Staubli VAL3: HIT_YD.pjx

--- HIT_YD.pjx ---
Parameters version=s7.6.2 stackSize=5000 millimeterUnit=true
Program file=OMAC_Abort.pgx
Program file=OMAC_Hold.pgx
Program file=OMAC_Main.pgx
Program file=OMAC_Reset.pgx
Program file=OMAC_Start.pgx
Program file=OMAC_Stop.pgx
Program file=OMAC_Unhold.pgx
Program file=blow.pgx
Program file=bypassPick.pgx
Program file=cellManager.pgx
Program file=getToolStatus.pgx
Program file=goHome.pgx
Program file=init.pgx
Program file=initTracking.pgx
Program file=isInSafetyArea.pgx
Program file=ModbusGet.pgx
Program file=modbusSet.pgx
Program file=overflowPick.pgx
Program file=Place.pgx
Program file=productionCycle.pgx
Program file=robot2PC.pgx
Program file=robot2PLC.pgx
Program file=send2NextRob.pgx
Program file=setAlarm.pgx
Program file=setConvSpeed.pgx
Program file=start.pgx
Program file=stop.pgx
Program file=trackErr_init.pgx
Program file=trackingPick.pgx
Program file=transferQueue.pgx
Data file=HIT_YD.dtx
Library alias=mot path=Disk://Tracking/Motion/Motion.pjx autoload=true password=
Type name=object path=Disk://Tracking/Templates/object/object.pjx

--- HIT_YD.dtx ---
aio aConvSpeed = {link=ModbusSrv-0\Modbus-Word\ao[3]}
aio aPlcCmd = {link=ModbusSrv-0\Modbus-Word\ai[0]}
aio aRbAlarm = {link=ModbusSrv-0\Modbus-Word\ao[0]}
aio aRbStatus = {link=ModbusSrv-0\Modbus-Word\ao[1]}
bool _bConvExist = true
bool _bEndCycle
bool _bIsPicking = true
bool _bIsPlacing
bool _bMutexCnvQueue = true
bool _bOverflowed = true
bool _bPartInTool
bool _bSentToHome = true
bool _bVisionOK = true
bool bLockPage
bool bPickDetection
bool bSetConvSpeed
bool bSyn
bool bTransferData = true
dio dAlarm[8]
  [0] = {link=ModbusSrv-0\Modbus-Bit\do[8]}
  [1] = {link=ModbusSrv-0\Modbus-Bit\do[9]}
  [2] = {link=ModbusSrv-0\Modbus-Bit\do[10]}
  [3] = {link=ModbusSrv-0\Modbus-Bit\do[11]}
  [4] = {link=ModbusSrv-0\Modbus-Bit\do[12]}
  [5] = {link=ModbusSrv-0\Modbus-Bit\do[13]}
  [6] = {link=ModbusSrv-0\Modbus-Bit\do[14]}
  [7] = {link=ModbusSrv-0\Modbus-Bit\do[15]}
dio dBlow = {link=BasicIO-1\%Q5}
dio dConvControl[2]
  [0] = {link=BasicIO-1\%I4}
  [1] = {link=BasicIO-1\%Q6}
dio dPartInTool = {link=fIn0}
dio dPermitPlace[4]
  [0] = {link=BasicIO-1\%I3}
  [1] = {link=BasicIO-1\%I2}
  [2] = {link=BasicIO-1\%I1}
  [3] = {link=BasicIO-1\%I0}
dio dPlaceDone[4]
  [0] = {link=BasicIO-1\%Q11}
  [1] = {link=BasicIO-1\%Q10}
  [2] = {link=BasicIO-1\%Q9}
  [3] = {link=BasicIO-1\%Q8}
dio dStartControl[4]
  [0] = {link=ModbusSrv-0\Modbus-Bit\di[4]}
  [1] = {link=ModbusSrv-0\Modbus-Bit\di[5]}
  [2] = {link=ModbusSrv-0\Modbus-Bit\di[6]}
  [3] = {link=ModbusSrv-0\Modbus-Bit\di[7]}
dio dStartState[4]
  [0] = {link=ModbusSrv-0\Modbus-Bit\do[4]}
  [1] = {link=ModbusSrv-0\Modbus-Bit\do[5]}
  [2] = {link=ModbusSrv-0\Modbus-Bit\do[6]}
  [3] = {link=ModbusSrv-0\Modbus-Bit\do[7]}
dio dVacuum = {link=BasicIO-1\%Q4}
frame fConveyor = {x=365.904087, y=326.91934, z=-82.602337, rx=-0.010861, ry=-0.059106, rz=0.004608, fatherId=world[0]}
frame fDetection = {x=392.598601, y=461.346273, z=-82.976862, rx=0.205045, ry=0.617271, rz=0.011036, fatherId=world[0]}
jointRs jDropPart = {j1=102.785955, j2=-95.43121, j3=69.578977, j4=134.260732}
jointRs jHome = {j1=102.785955, j2=-95.43121, j3=69.578977, j4=134.260732}
jointRs jPark = {j1=102.785955, j2=-95.43121, j3=69.578977, j4=134.260732}
mdesc _mLoad = {accel=98.01, vel=99, decel=98.01, leave=40, reach=40}
mdesc mLoad = {accel=121, vel=110, decel=121, leave=40, reach=40}
mdesc mNomSpeed = {accel=121, vel=110, decel=121, leave=20, reach=20}
mdesc mPickDown = {accel=144, vel=120, decel=144, blend=off, leave=10, reach=10}
mdesc mPickup = {accel=121, vel=110, decel=121, leave=40, reach=40}
mdesc mPlaceDown = {accel=144, vel=120, decel=144, blend=off, leave=15, reach=15}
mdesc mPlaceUp = {accel=169, vel=130, decel=169, blend=cartesian, leave=30, reach=30}
mdesc mSlow = {accel=1, vel=10, decel=1, leave=10, reach=10}
mdesc mUnload = {accel=121, vel=110, decel=121, leave=40, reach=40}
num _nBlowDelay
num _nCntBypassed = 1
num _nCntPartsDone[2]
  [0] = 234927
  [1] = 234852
num _nCntTransfered = 2732
num _nConvSpd = 482.240758
num _nCycleTime[4]
  [0] = 2.619
  [1] = 0.715
  [2] = 2.425
  [3] = 0.561
num _nCycleTimeIndx = 2
num _nID = 1
num _nLastStateCMD
num _nOmacStat = 3
num _nPartID = 1
num _nPlaceCurItem[2]
num _nPullIndexTQ = 32
num _nPushIndexTQ = 32
num _nStateCMD
num _nTimer = 6773.495
num _nTrackErr = 334
num nBlowID = 0.4
num nBypass = 1
num nLoadRatio[4]
  [0] = 0.85
  [1] = 0.9
  [2] = 0.9
  [3] = 1
num nNomConvSpeed = 100
num nPartHeight = 5
num nPickAppro = 65
num nPickOS_X
num nPickOS_Y = 2
num nPlaceAppro = 60
public num nPlaceNum
num nSafeMaxX = 850
num nSafeMaxY = 650
num nSafeMinX
num nSafeMinY
num nStopTime
num nTestData[5]
  [0] = 6
  [1] = -49
  [2] = 55
  [4] = 184151
num nVacuumID = 0.1
num nWaitDist2Up4BP = -300
num nWaitDistToDown = 50
num nWaitDistToUp[1 3]
  [0,0] = -80
  [0,1] = 120
  [0,2] = 400
num nWaitDistX
object _oTransferQueue[1 100]
  [0,0]
    num nID = -1
    num nLatchedValue
    trsf trTrsf
  [0,1]
    num nID = -1
    num nLatchedValue
    trsf trTrsf
  [0,2]
    num nID = -1
    num nLatchedValue
    trsf trTrsf
  [0,3]
    num nID = -1
    num nLatchedValue
    trsf trTrsf
  [0,4]
    num nID = -1
    num nLatchedValue
    trsf trTrsf
  [0,5]
    num nID = -1
    num nLatchedValue
    trsf trTrsf
  [0,6]
    num nID = -1
    num nLatchedValue
    trsf trTrsf
  [0,7]
    num nID = -1
    num nLatchedValue
    trsf trTrsf
  [0,8]
    num nID = -1
    num nLatchedValue
    trsf trTrsf
  [0,9]
    num nID = -1
    num nLatchedValue
    trsf trTrsf
  [0,10]
    num nID = -1
    num nLatchedValue
    trsf trTrsf
  [0,11]
    num nID = -1
    num nLatchedValue
    trsf trTrsf
  [0,12]
    num nID = -1
    num nLatchedValue
    trsf trTrsf
  [0,13]
    num nID = -1
    num nLatchedValue
    trsf trTrsf
  [0,14]
    num nID = -1
    num nLatchedValue
    trsf trTrsf
  [0,15]
    num nID = -1
    num nLatchedValue
    trsf trTrsf
  [0,16]
    num nID = -1
    num nLatchedValue
    trsf trTrsf
  [0,17]
    num nID = -1
    num nLatchedValue
    trsf trTrsf
  [0,18]
    num nID = -1
    num nLatchedValue
    trsf trTrsf
  [0,19]
    num nID = -1
    num nLatchedValue
    trsf trTrsf
  [0,20]
    num nID = -1
    num nLatchedValue
    trsf trTrsf
  [0,21]
    num nID = -1
    num nLatchedValue
    trsf trTrsf
  [0,22]
    num nID = -1
    num nLatchedValue
    trsf trTrsf
  [0,23]
    num nID = -1
    num nLatchedValue
    trsf trTrsf
  [0,24]
    num nID = -1
    num nLatchedValue
    trsf trTrsf
  [0,25]
    num nID = -1
    num nLatchedValue
    trsf trTrsf
  [0,26]
    num nID = -1
    num nLatchedValue
    trsf trTrsf
  [0,27]
    num nID = -1
    num nLatchedValue
    trsf trTrsf
  [0,28]
    num nID = -1
    num nLatchedValue
    trsf trTrsf
  [0,29]
    num nID = -1
    num nLatchedValue
    trsf trTrsf
  [0,30]
    num nID = -1
    num nLatchedValue
    trsf trTrsf
  [0,31]
    num nID = -1
    num nLatchedValue
    trsf trTrsf
  [0,32]
    num nID = -1
    num nLatchedValue
    trsf trTrsf
  [0,33]
    num nID = -1
    num nLatchedValue
    trsf trTrsf
  [0,34]
    num nID = -1
    num nLatchedValue
    trsf trTrsf
  [0,35]
    num nID = -1
    num nLatchedValue
    trsf trTrsf
  [0,36]
    num nID = -1
    num nLatchedValue
    trsf trTrsf
  [0,37]
    num nID = -1
    num nLatchedValue
    trsf trTrsf
  [0,38]
    num nID = -1
    num nLatchedValue
    trsf trTrsf
  [0,39]
    num nID = -1
    num nLatchedValue
    trsf trTrsf
  [0,40]
    num nID = -1
    num nLatchedValue
    trsf trTrsf
  [0,41]
    num nID = -1
    num nLatchedValue
    trsf trTrsf
  [0,42]
    num nID = -1
    num nLatchedValue
    trsf trTrsf
  [0,43]
    num nID = -1
    num nLatchedValue
    trsf trTrsf
  [0,44]
    num nID = -1
    num nLatchedValue
    trsf trTrsf
  [0,45]
    num nID = -1
    num nLatchedValue
    trsf trTrsf
  [0,46]
    num nID = -1
    num nLatchedValue
    trsf trTrsf
  [0,47]
    num nID = -1
    num nLatchedValue
    trsf trTrsf
  [0,48]
    num nID = -1
    num nLatchedValue
    trsf trTrsf
  [0,49]
    num nID = -1
    num nLatchedValue
    trsf trTrsf
  [0,50]
    num nID = -1
    num nLatchedValue
    trsf trTrsf
  [0,51]
    num nID = -1
    num nLatchedValue
    trsf trTrsf
  [0,52]
    num nID = -1
    num nLatchedValue
    trsf trTrsf
  [0,53]
    num nID = -1
    num nLatchedValue
    trsf trTrsf
  [0,54]
    num nID = -1
    num nLatchedValue
    trsf trTrsf
  [0,55]
    num nID = -1
    num nLatchedValue
    trsf trTrsf
  [0,56]
    num nID = -1
    num nLatchedValue
    trsf trTrsf
  [0,57]
    num nID = -1
    num nLatchedValue
    trsf trTrsf
  [0,58]
    num nID = -1
    num nLatchedValue
    trsf trTrsf
  [0,59]
    num nID = -1
    num nLatchedValue
    trsf trTrsf
  [0,60]
    num nID = -1
    num nLatchedValue
    trsf trTrsf
  [0,61]
    num nID = -1
    num nLatchedValue
    trsf trTrsf
  [0,62]
    num nID = -1
    num nLatchedValue
    trsf trTrsf
  [0,63]
    num nID = -1
    num nLatchedValue
    trsf trTrsf
  [0,64]
    num nID = -1
    num nLatchedValue
    trsf trTrsf
  [0,65]
    num nID = -1
    num nLatchedValue
    trsf trTrsf
  [0,66]
    num nID = -1
    num nLatchedValue
    trsf trTrsf
  [0,67]
    num nID = -1
    num nLatchedValue
    trsf trTrsf
  [0,68]
    num nID = -1
    num nLatchedValue
    trsf trTrsf
  [0,69]
    num nID = -1
    num nLatchedValue
    trsf trTrsf
  [0,70]
    num nID = -1
    num nLatchedValue
    trsf trTrsf
  [0,71]
    num nID = -1
    num nLatchedValue
    trsf trTrsf
  [0,72]
    num nID = -1
    num nLatchedValue
    trsf trTrsf
  [0,73]
    num nID = -1
    num nLatchedValue
    trsf trTrsf
  [0,74]
    num nID = -1
    num nLatchedValue
    trsf trTrsf
  [0,75]
    num nID = -1
    num nLatchedValue
    trsf trTrsf
  [0,76]
    num nID = -1
    num nLatchedValue
    trsf trTrsf
  [0,77]
    num nID = -1
    num nLatchedValue
    trsf trTrsf
  [0,78]
    num nID = -1
    num nLatchedValue
    trsf trTrsf
  [0,79]
    num nID = -1
    num nLatchedValue
    trsf trTrsf
  [0,80]
    num nID = -1
    num nLatchedValue
    trsf trTrsf
  [0,81]
    num nID = -1
    num nLatchedValue
    trsf trTrsf
  [0,82]
    num nID = -1
    num nLatchedValue
    trsf trTrsf
  [0,83]
    num nID = -1
    num nLatchedValue
    trsf trTrsf
  [0,84]
    num nID = -1
    num nLatchedValue
    trsf trTrsf
  [0,85]
    num nID = -1
    num nLatchedValue
    trsf trTrsf
  [0,86]
    num nID = -1
    num nLatchedValue
    trsf trTrsf
  [0,87]
    num nID = -1
    num nLatchedValue
    trsf trTrsf
  [0,88]
    num nID = -1
    num nLatchedValue
    trsf trTrsf
  [0,89]
    num nID = -1
    num nLatchedValue
    trsf trTrsf
  [0,90]
    num nID = -1
    num nLatchedValue
    trsf trTrsf
  [0,91]
    num nID = -1
    num nLatchedValue
    trsf trTrsf
  [0,92]
    num nID = -1
    num nLatchedValue
    trsf trTrsf
  [0,93]
    num nID = -1
    num nLatchedValue
    trsf trTrsf
  [0,94]
    num nID = -1
    num nLatchedValue
    trsf trTrsf
  [0,95]
    num nID = -1
    num nLatchedValue
    trsf trTrsf
  [0,96]
    num nID = -1
    num nLatchedValue
    trsf trTrsf
  [0,97]
    num nID = -1
    num nLatchedValue
    trsf trTrsf
  [0,98]
    num nID = -1
    num nLatchedValue
    trsf trTrsf
  [0,99]
    num nID = -1
    num nLatchedValue
    trsf trTrsf
pointRs pPick = {x=51.000306, y=-30.000014, z=4.992462, rx=0, ry=0, rz=112.9, shoulder=lefty, fatherId=fDetection[0]}
pointRs pPlace[4]
  [0] = {x=360, y=110, z=-83, rx=180, ry=0, rz=-100, shoulder=lefty, fatherId=world[0]}
  [1] = {x=490, y=105, z=-83, rx=180, ry=0, rz=-100, shoulder=lefty, fatherId=world[0]}
  [2] = {x=620, y=105, z=-83, rx=180, rz=-98.02183, shoulder=lefty, fatherId=world[0]}
  [3] = {x=760, y=105, z=-83, rx=180, rz=-98.02084, shoulder=lefty, fatherId=world[0]}
sio skToRobot = {link=Socket\toRobot_sk1}
sio sktoPC = {link=Socket\toPC}
sio synServer = {link=Socket\synRobot1}
string _sCycleStatus = "Distance to pick: -359.23"
string sConveyorList = "cvIn"
string sDataPC = "run"
string sString = "done"
tool tGripper = {z=85, rz=45, fatherId=flange[0], ioLink=valve1}

--- start.pgx ---
program start()
begin
  //
  cls()
  userPage()
  put("Running...")
  //
  //1.-  Make sure that the hardware is working:
  //     a)  The encoder counts are increasing when the conveyor is moving forward.
  //     b)  The controller trigger output is seen by the encoder input interface (exxLatchSig input on a Dual ABZ board) and by the vision system.
  //2.-  Define TCP Sockets:
  //     a)  TCP Client “cognex1”  (port 1023 to camera's IP address)
  //     b)  TCP Client “toRobot_sk1” (port 1001 to next robot IP address)
  //     c)  TCP Client “toRobot_sk2” (port 1002 to next robot IP address)
  //     d)  TCP Server “fromRobot_sk1” (port 1001)
  //     e)  TCP Server “fromRobot_sk2” (port 1002)
  //3.-  Use the Wizard to create two new conveyors library (F6)
  //4.-  Use the Wizard to define the settings for the conveyors libraries (F7)
  //5.-  Use the Wizard to define the scale factor and the conveyor geometry of each conveyor(F1)
  //6.-  Use the Wizard to calibrate the vision frame of each conveyor (F4)
  //7.-  Check that the program detection() from the library Tracking\Detections\Cognex search the results on the right cell of the cognex spreadsheet
  //8.-  Enter the name of you conveyors libraries in the sConveyorList string variable.
  //9.-  Define your tool and teach the jDropPart, jHome, jPark positions.
  //10.- Run the application.
  //
  //
  userPage(bLockPage)
  call init()

  // General managment
  taskCreate "isInSafetyArea",100,isInSafetyArea()
  call OMAC_Main()
end

--- init.pgx ---
program init()
  local num l_nI
  local num l_nJ
begin
  // This program initialize all variables
  //
  // Input parameters
  //  None            :
  //
  // Output parameters
  //  None            :
  //
  //----------------------------------------------------------------
  //
  //che add
  nPlaceNum=3
  sDataPC="stop"


  // Booleans
  _bSentToHome=false
  _bMutexCnvQueue[0]=false
  _bIsPicking=false
  _bIsPlacing=false
  _bConvExist=false
  _bEndCycle=false
  //

  //
  // Numerical
  _nBlowDelay=0
  _nID[0]=-1
  _nCntBypassed[0]=0
  //_nCntBypassed[0]=nBypass[0]
  _nCntTransfered[0]=0

  _nPushIndexTQ[0]=0
  _nPullIndexTQ[0]=0
  _nTimer=0

  resize(_nCycleTime,1,4)
  for _nCycleTimeIndx=0 to size(_nCycleTime)-1
    _nCycleTime[_nCycleTimeIndx]=0
  endFor
  _nCycleTimeIndx=0

  //dio
  dPlaceDone[0]=false
  dPlaceDone[1]=false
  dPlaceDone[2]=false
  dPlaceDone[3]=false

  // aio
  aioSet(aRbAlarm,0)
  //call setAlarm(0)
  clearBuffer(synServer)
  // Points
  pPick.trsf={0,0,0,0,0,0}

  //

  //
  // Transfer Queues
  for l_nI=0 to size(_oTransferQueue,2)-1
    _oTransferQueue[0,l_nI].nID=-1
    _oTransferQueue[0,l_nI].trTrsf={0,0,0,0,0,0}
    _oTransferQueue[0,l_nI].nLatchedValue=0
  endFor
  //
  // Strings
  _sCycleStatus=""
  autoConnectMove(true)
end

--- isInSafetyArea.pgx ---
program isInSafetyArea()
  local jointRs l_jHere
  local num l_ns
  local pointRs l_pCurrent
begin
  do
    l_pCurrent=here(flange,world)
    //**************************************************//
    //******** 用来判断机器人是否在安全工作空间 ********//
    //**************************************************//
    if (l_pCurrent.trsf.y>=nSafeMaxY or l_pCurrent.trsf.y<=nSafeMinY or l_pCurrent.trsf.x>=nSafeMaxX or l_pCurrent.trsf.x<=nSafeMinX) and _nOmacStat==3
      aioSet(aRbAlarm,10)
      call setAlarm(7)
      popUpMsg("机器人超出安全工作空间！")
      logMsg("机器人超出安全工作空间！")
      call OMAC_Abort()
    endIf

    if (dConvControl[0]==true)
      dConvControl[1]=true
    else
      dConvControl[1]=false
    endIf
    delay(0)
  until false
end

--- ModbusGet.pgx ---
program modbusGet(num& x_nResult (dimensions=1))
begin
  //start
  if (dStartControl[1]==true and dStartControl[2]==false and dStartControl[3]==false)
    x_nResult=1
    //stop
  elseIf (dStartControl[1]==false and dStartControl[2]==true and dStartControl[3]==false)
    x_nResult=2
    //reset
  elseIf (dStartControl[1]==false and dStartControl[2]==false and dStartControl[3]==true)
    x_nResult=3
    //other
  else
    x_nResult=0
  endIf
end

--- OMAC_Hold.pgx ---
program OMAC_Hold()
  local joint l_jHere
begin
  //OMAC进程:Holding
  _nOmacStat=5
  logMsg("上位机手动操作：暂停")
  _bEndCycle=true
  wait(taskStatus("productionCycle")==-1)
  _bMutexCnvQueue[0]=false
  taskKill("cellManager")
  wait(taskStatus("cellManager")==-1)
  stopMove()
  resetMotion()
  // Move up axis 3
  l_jHere=herej()
  l_jHere.j3=95
  movej(l_jHere,tGripper,mSlow)
  movej(jHome,tGripper,mSlow)
  waitEndMove()
  disablePower()
  dVacuum=false
  wait(isSettled())
  wait(isPowered()==false)
  //OMAC进程:Held
  _nOmacStat=6
  delay(0)
end

--- OMAC_Main.pgx ---
program OMAC_Main()
begin
  //  _nOmacStat
  //1-Ready
  //2-Starting
  //3-Running
  //4-Resetting
  //5-Holding
  //6-Held
  //7-Un-Holding
  //8-Stopping
  //9-Stopped
  //10-Aborting


  // _nStateCmd
  //1-Start
  //2-Stop
  //3-Reset
  //4-Hold
  //10-Abort

  //机器人状态
  _nOmacStat=9

  _nLastStateCMD=0
  //OMAC_init
  call init()
  do
    switch _nOmacStat
      //复位信号
      case 1
        call modbusSet(3)
      break
      //运行信号
      case 3
        call modbusSet(1)
      break
      //准备信号
      case 4
        call modbusSet(2)
      break
      //停止信号
      case 9
        call modbusSet(2)
      break
      default
      break
    endSwitch


    //机器人状态输出
    //call modbusSet(_nOmacStat)
    //aioSet(aRbStatus,_nOmacStat)
    //根据上位机按钮转换为指令num
    //10-Abort
    if esStatus()==2
      _nStateCMD=10
    else
      //_nStateCMD=aioGet(aPlcCmd)
      call modbusGet(_nStateCMD)
    endIf

    //根据指令num，触发相应动作
    if _nStateCMD!=_nLastStateCMD
      switch _nStateCMD
        //Reset
        case 3
          //确认当前OMAC进程为stopped
          if _nOmacStat==9

            if taskStatus("Reset")>=0
              taskKill("Reset")
            endIf
            wait(taskStatus("Reset")<0)
            taskCreate "Reset",100,OMAC_Reset()

          endIf
        break

        //Start
        case 1
          //确认当前OMAC进程为Ready
          if _nOmacStat==1

            if taskStatus("Start")>=0
              taskKill("Start")
            endIf
            wait(taskStatus("Start")<0)
            taskCreate "Start",100,OMAC_Start()

          elseIf _nOmacStat==6
            //确认当前OMAC进程为Held

            if taskStatus("Unhold")>=0
              taskKill("Unhold")
            endIf
            wait(taskStatus("Unhold")<0)
            taskCreate "Unhold",100,OMAC_Unhold()
          else
            //call setAlarm(7)

          endIf
        break
        //Hold
        case 4
          //确认当前OMAC进程为running
          if _nOmacStat==3

            if taskStatus("Hold")>=0
              taskKill("Hold")
            endIf
            wait(taskStatus("Hold")<0)
            taskCreate "Hold",100,OMAC_Hold()

          endIf
        break

        //Unhold
        case 7

        break

        //Stop
        case 2
          //确认当前OMAC进程不是停止
          if _nOmacStat!=9
            if taskStatus("Stop")>=0
              taskKill("Stop")
            endIf
            wait(taskStatus("Stop")<0)
            taskCreate "Stop",100,OMAC_Stop()
          endIf
        break

        //Abort
        case 10
          // //确认当前OMAC进程不是停止
          if _nOmacStat!=9
            if taskStatus("Abort")>=0
              taskKill("Abort")
            endIf
            wait(taskStatus("Abort")<0)
            taskCreate "Abort",100,OMAC_Abort()
          endIf
        break

      endSwitch
    endIf
    //记录上次指令
    _nLastStateCMD=_nStateCMD
    delay(0)
  until false


end

--- OMAC_Reset.pgx ---
program OMAC_Reset()
  local bool l_bResult
  local joint l_jHere
  local num l_nKey
begin

  //OMAC进程:resetting
  _nOmacStat=4
  logMsg("上位机手动操作：复位")



  // Reset conveyor speed
  //  call setConvSpeed(0,0)
  //start vision
  _bVisionOK=false
  if taskStatus("robot2PC")>=0
    taskKill("robot2PC")
  endIf
  wait(taskStatus("robot2PC")<0)
  taskCreate "robot2PC",100,robot2PC()
  //wait vision ok
  l_bResult=watch(_bVisionOK,5)
  if l_bResult==false
    //alarm
    call setAlarm(0)
    logMsg("vision start failed")
    taskKill("robot2PC")
    _nOmacStat=9
    return
  endIf
  // Variable initializing
  call init()
  call trackErr_init()
  // Launch Tracking
  call initTracking()
  if !isInRange(herej())
    aioSet(aRbAlarm,20)
    call setAlarm(1)
    popUpMsg("机器人关节超限!")
    taskCreate "Abort",100,OMAC_Abort()
    return
  endIf
  //
  resetMotion()
  // Enables arm power
  while !isPowered()
    enablePower()
    delay(1)
  endWhile
  _bSentToHome=true
  // Send robot to home position
  l_jHere=herej()
  l_jHere.j3=jHome.j3
  movej(l_jHere,tGripper,mSlow)
  movej(jHome,tGripper,mSlow)
  //
  //
  // Init user screen
  cls()
  gotoxy(0,4)
  put("Cycle Time (Last):    ")
  gotoxy(0,6)
  put("Cycle Time (Average): ")
  gotoxy(0,8)
  put("Cycle Time (Best):    ")
  gotoxy(0,10)
  put("      Pick                Place         ")
  gotoxy(0,11)
  put("  Done   Transfer      Done   ")


  //Launch queue transfer tasks
  if bTransferData[0]
    if taskStatus("TransferQueue1")>=0
      taskKill("TransferQueue1")
    endIf
    taskCreate "TransferQueue1",100,transferQueue(0)
    wait(taskStatus("TransferQueue1")==1)
  endIf

  // Task to remove picking positions that have pass the downstream limit while the robot is placing a part.
  if taskStatus("overflowPick")>=0
    taskKill("overflowPick")
  endIf
  taskCreate "overflowPick",100,overflowPick()
  wait(taskStatus("overflowPick")==1)

  //OMAC进程:ready
  _nOmacStat=1
  delay(0)
end

--- Place.pgx ---
program place()
  local bool l_bNoError
  local joint l_jAppro
  local num l_nConvNum
  local num l_nError
  local num l_nMoveID
  local num l_nTrackStatus
  local pointRs l_pAppro
  local pointRs l_pPlace
  local string l_sToolStatus
begin
  l_nConvNum=1
  link(l_pPlace,world)
  //che modify start
  if nPlaceNum<0
    nPlaceNum=3
  endIf
  _mLoad=mLoad
  _mLoad.vel=mLoad.vel*nLoadRatio[nPlaceNum]
  _mLoad.accel=mLoad.accel*nLoadRatio[nPlaceNum]*nLoadRatio[nPlaceNum]
  _mLoad.decel=mLoad.decel*nLoadRatio[nPlaceNum]*nLoadRatio[nPlaceNum]

  //dControlVacuum[nPlaceNum]=false
  l_pPlace=pPlace[nPlaceNum]
  //end
  // Place part
  l_pAppro=appro(l_pPlace,{0,0,-nPlaceAppro,0,0,0})
  l_bNoError=pointToJoint(tGripper,jHome,l_pAppro,l_jAppro)
  call mot:getTrackStatus(l_nTrackStatus)
  if l_nTrackStatus>0
    // Use trackOff if the robot is synchronized
    if l_bNoError
      call mot:trackOffJ(l_jAppro,tGripper,_mLoad,l_nMoveID,l_nError)
    else
      call mot:trackOff(l_pAppro,tGripper,_mLoad,l_nMoveID,l_nError)
    endIf
  else
    // Use movej if the robot is not synchronized
    if l_bNoError
      l_nMoveID=movej(l_jAppro,tGripper,_mLoad)
    else
      l_nMoveID=movej(l_pAppro,tGripper,_mLoad)
    endIf
  endIf
  // wait permit signal
  //
  wait(dPermitPlace[nPlaceNum]==true)
  l_nMoveID=movel(l_pPlace,tGripper,mPlaceDown)
  wait(getMoveId()>l_nMoveID+nBlowID)
  _nBlowDelay=0.2
  waitEndMove()
  //delay(nStopTime)
  l_nMoveID=movel(l_pAppro,tGripper,mPlaceUp)
  // check PartInTool if bPickDetection
  if bPickDetection
    //wait(getMoveId()>l_nMoveID-0.8)
    wait(getMoveId()>l_nMoveID+nBlowID-1.2)
    call getToolStatus(l_sToolStatus)
  else
    //wait(getMoveId()>l_nMoveID-0.2)
    wait(getMoveId()>l_nMoveID+nBlowID-1.2)
    _bPartInTool=false
  endIf
  // send done signal
  //dPlaceDone[nPlaceNum]=true
  wait(getMoveId()>l_nMoveID+0.1)
  delay(0)
  //dPlaceDone[nPlaceNum]=false
  if l_sToolStatus=="PartInTool" or _bPartInTool==false
    // A part has been placed
    _nCntPartsDone[l_nConvNum]=_nCntPartsDone[l_nConvNum]+1
  endIf
  delay(0)

  dPlaceDone[nPlaceNum]=true
  wait(getMoveId()>l_nMoveID+0.4)
  if nPlaceNum==3 and bSyn
    do
      sString=synServer
    until (sString=="done")
  endIf
  if nPlaceNum==0
    //synServer="done"
  endIf
  nPlaceNum=nPlaceNum-1
  nTestData[4]=nTestData[4]+1
  //end

end

--- robot2PC.pgx ---
program robot2PC()
begin
  //清空缓存
  clearBuffer(sktoPC)
  //设置终止符 $
  sioCtrl(sktoPC,"endOfString",36)
  do
    sktoPC="run"
    sDataPC=sktoPC
    _bVisionOK=true
    delay(1)
  until false
end

--- setAlarm.pgx ---
program setAlarm(num x_nNum (dimensions=1))
  local num l_ns
begin
  switch x_nNum
    case 0
      dAlarm[0]=true
      dAlarm[1]=false
      dAlarm[2]=false
      dAlarm[3]=false
      dAlarm[4]=false
      dAlarm[5]=false
      dAlarm[6]=false
      dAlarm[7]=false
      delay(0.35)
      dAlarm[0]=false
      dAlarm[1]=false
      dAlarm[2]=false
      dAlarm[3]=false
      dAlarm[4]=false
      dAlarm[5]=false
      dAlarm[6]=false
      dAlarm[7]=false
    break
    case 1
      dAlarm[0]=false
      dAlarm[1]=true
      dAlarm[2]=false
      dAlarm[3]=false
      dAlarm[4]=false
      dAlarm[5]=false
      dAlarm[6]=false
      dAlarm[7]=false
      delay(0.35)
      dAlarm[0]=false
      dAlarm[1]=false
      dAlarm[2]=false
      dAlarm[3]=false
      dAlarm[4]=false
      dAlarm[5]=false
      dAlarm[6]=false
      dAlarm[7]=false
    break
    case 2
      dAlarm[0]=false
      dAlarm[1]=false
      dAlarm[2]=true
      dAlarm[3]=false
      dAlarm[4]=false
      dAlarm[5]=false
      dAlarm[6]=false
      dAlarm[7]=false
      delay(0.35)
      dAlarm[0]=false
      dAlarm[1]=false
      dAlarm[2]=false
      dAlarm[3]=false
      dAlarm[4]=false
      dAlarm[5]=false
      dAlarm[6]=false
      dAlarm[7]=false
    break
    case 3
      dAlarm[0]=false
      dAlarm[1]=false
      dAlarm[2]=true
      dAlarm[3]=false
      dAlarm[4]=false
      dAlarm[5]=false
      dAlarm[6]=false
      dAlarm[7]=false
      delay(0.35)
      dAlarm[0]=false
      dAlarm[1]=false
      dAlarm[2]=false
      dAlarm[3]=false
      dAlarm[4]=false
      dAlarm[5]=false
      dAlarm[6]=false
      dAlarm[7]=false
    break
    case 4
      dAlarm[0]=false
      dAlarm[1]=false
      dAlarm[2]=false
      dAlarm[3]=false
      dAlarm[4]=true
      dAlarm[5]=false
      dAlarm[6]=false
      dAlarm[7]=false
      delay(0.35)
      dAlarm[0]=false
      dAlarm[1]=false
      dAlarm[2]=false
      dAlarm[3]=false
      dAlarm[4]=false
      dAlarm[5]=false
      dAlarm[6]=false
      dAlarm[7]=false
    break
    case 5
      dAlarm[0]=false
      dAlarm[1]=false
      dAlarm[2]=false
      dAlarm[3]=false
      dAlarm[4]=false
      dAlarm[5]=true
      dAlarm[6]=false
      dAlarm[7]=false
      delay(0.35)
      dAlarm[0]=false
      dAlarm[1]=false
      dAlarm[2]=false
      dAlarm[3]=false
      dAlarm[4]=false
      dAlarm[5]=false
      dAlarm[6]=false
      dAlarm[7]=false
    break
    case 6
      dAlarm[0]=false
      dAlarm[1]=false
      dAlarm[2]=false
      dAlarm[3]=false
      dAlarm[4]=false
      dAlarm[5]=false
      dAlarm[6]=true
      dAlarm[7]=false
      delay(0.35)
      dAlarm[0]=false
      dAlarm[1]=false
      dAlarm[2]=false
      dAlarm[3]=false
      dAlarm[4]=false
      dAlarm[5]=false
      dAlarm[6]=false
      dAlarm[7]=false
    break
    case 7
      dAlarm[0]=false
      dAlarm[1]=false
      dAlarm[2]=false
      dAlarm[3]=false
      dAlarm[4]=false
      dAlarm[5]=false
      dAlarm[6]=false
      dAlarm[7]=true
      delay(0.35)
      dAlarm[0]=false
      dAlarm[1]=false
      dAlarm[2]=false
      dAlarm[3]=false
      dAlarm[4]=false
      dAlarm[5]=false
      dAlarm[6]=false
      dAlarm[7]=false
    break
    default
      dAlarm[0]=false
      dAlarm[1]=false
      dAlarm[2]=false
      dAlarm[3]=false
      dAlarm[4]=false
      dAlarm[5]=false
      dAlarm[6]=false
      dAlarm[7]=false
    break
  endSwitch
end

--- stop.pgx ---
program stop()
  local joint l_jHere
  local string l_sToolStatus
begin
  //
  l_sToolStatus=""
  //
  cls()
  gotoxy(10,6)
  put("Application Ending")
  //
  stopMove()
  resetMotion()
  disablePower()
  // Stop all tasks
  taskKill("TransferQueue1")
  taskKill("overflowPick")
  taskKill("productionCycle")
  taskKill("blow")
  taskKill("changePallet")
  taskKill("isInSafetyArea")
  taskKill("robot2PC")
  taskKill("robot2PLC")

  if _bConvExist
    call mot:kill()
  endIf

  //
  // Stop conveyor speed
  call setConvSpeed(0,0)
  //
  // Reset triggers
  //  dioSet(dTrigger,0)
  //
  resetMotion()
  //
  //
  // Move up axis 3
  l_jHere=herej()
  l_jHere.j3=90
  //movej(l_jHere,flange,mSlow)
  //
  // Drop the part on the tool
  if bPickDetection
    call getToolStatus(l_sToolStatus)
  endIf
  if l_sToolStatus=="PartInTool" or !bPickDetection
    //movej(jDropPart,flange,mSlow)
    //waitEndMove()
    dBlow=true
    dVacuum=false
    delay(0.5)
    dBlow=false
  else
    dVacuum=false
    dBlow=false
  endIf
  //
  // Go to park position
  //movej(jPark,flange,mSlow)
  //waitEndMove()
  disablePower()
  //
  cls()
  gotoxy(10,6)
  put("Application Ended")
  //
end
